FUNCTION_BLOCK FB_Observable_UINT EXTENDS FB_AbstractObservable
VAR
    _nVal:              UINT;
    _nOldVal:           UINT;
END_VAR

METHOD FB_init : BOOL
VAR_INPUT
    bInitRetains:       BOOL; // if TRUE, the retain variables are initialized (warm start / cold start)
    bInCopyCode:        BOOL;  // if TRUE, the instance afterwards gets moved into the copy code (online change)
END_VAR
THIS^._nTypeClass := __SYSTEM.TYPE_CLASS.TYPE_UINT;
END_METHOD

PROPERTY nDataSize : UDINT
GET
nDataSize := SIZEOF(UINT);
END_GET
END_PROPERTY

PROPERTY nValue16 : UINT
GET
nValue16 := THIS^._nVal;
END_GET
SET
THIS^._nOldVal := THIS^._nVal;
THIS^._nVal := nValue16;

THIS^.NotifyWithConditions();
END_SET
END_PROPERTY

PROPERTY PROTECTED pData : POINTER TO BYTE
GET
pData := ADR(THIS^._nVal);
END_GET
END_PROPERTY

METHOD  ValueChanged : BOOL
VAR_INPUT
END_VAR
ValueChanged := THIS^._nOldVal <> THIS^._nVal;
END_METHOD

END_FUNCTION_BLOCK

(* stored: Version 1.1.0.1, ProductVersion 3.1.4024.12
   POU FB_Observable_UINT: Id {f2d7fe92-4d1e-47f3-bc2f-43e40068362f}, SpecialFunc None
   Method FB_init: Id {a8d1dafc-ecc5-0651-0bc9-0243a5da7a8f}
   Property nDataSize: Id {10d98ff7-fb78-4548-99e7-5a2a26b39e70}
   Get Get: Id {27478cea-7c50-4fe9-ad87-127a0ce7570c}
   Property nValue16: Id {af502dac-a26d-48ef-8a2d-4ee091e8d385}
   Get Get: Id {f747421d-9861-4e67-82a8-164d0b8556a2}
   Set Set: Id {1715d78f-c08f-4f38-91ae-928e9c0a47c7}
   Property pData: Id {ff871db6-7dd8-4611-acda-6b03ac39c9ac}
   Get Get: Id {63c9fd73-b318-4041-b3a2-bd5445f39df2}
   Method ValueChanged: Id {0f03086f-698e-00fd-3ab2-3bf86cc1a756} *)
